// TIA Portal V17 export
// export: Created 2023-12-22T15:05:35.8060205Z, ExportSetting WithDefaults, DisplayName Totally Integrated Automation Portal, DisplayVersion V17, DisplayName TIA Portal Openness, DisplayVersion V17, DisplayName TIA Portal Version Control Interface, DisplayVersion V17, DisplayName STEP 7 Professional, DisplayVersion V17, DisplayName STEP 7 Safety, DisplayVersion V17, DisplayName WinCC Advanced, DisplayVersion V17
TYPE "PolyMix_Output"
// stored: IsFailsafeCompliant false
   STRUCT
      WatchDog : Int;
      Clock : Bool;
      Start : Bool;   // Установка в работе
      LS_1 : Bool;   // РУ-1
      LS_2 : Bool;   // РУ-2
      LS_3 : Bool;   // РУ-3
      LS_4 : Bool;   // РУ-4
      KC_1 : Bool;   // Статус клапана КС-1
      ALLS : Bool;   // Аварийно низкий уровень
      Local : Bool;   // 0 - местный режим, 1 - дистанционный
      LLS : Bool;   // Низкий уровень в полимиксе
      HLS : Bool;   // Высокий уровен в полимиксе
      SP_C : Real;   // Заданная концентрация
      Level : Real;   // Уровень в баке
      Flow : Real;   // Скорость потока
      Weight : Real;
      Mix_1 : Int;   // Статус М1
      Mix_2 : Int;   // Статус М2
      Mix_3 : Int;   // Статус М3
      SD : Int;   // Статус ШД
      DD : Int;   // Статус ЧП
      SH : Int;   // Статус ТШ
      PN : Int;   // Статус ПТ
      Vibro : Int;   // Статус вибратора
      Vent : Int;   // Статус вентилятора
      Messages : Struct   // - Аварийные сообщения
         Flow_Dry_Run : Bool;   // Авария - нет протока КС-1
         Flow_Low : Bool;   // Авария - низкий проток КС-1
         LE_NoChange : Bool;   // Авария - не заполняется бак
         LE_Low : Bool;   // Авария - низкий уровень в баке
         LE_High : Bool;   // Авария - высокий уровень в баке
         LS_Low : Bool;   // Авария - низкий уровень в буфере
         LS_NoProduct : Bool;   // Авария - нет продукта в бункере
         LS_Filter : Bool;   // Авария - полный бункер
         SD_Low : Bool;   // Авария - низкая скорость дозации
         Low_Weight : Bool;   // Авария - мало продукта в бункере
         Link_Error : Bool;   // Предупреждение - нет связи со шкафов дозации
         Alarm : Word;   // Слово аварий для панели
      END_STRUCT;
      Report : "PolyMix_Report";   // Отчёт за вчера
      LE_Alarm { S7_SetPoint := 'True'} : Word;   // Слово аврарий датчика уровня
   END_STRUCT;
END_TYPE
